// TIA Portal project "FactoryIO_Template_S7-1200_V14" (V14)
// Vorlageprojekt für das Buch mit Zielsystem S7-1200

(* hardware
DEVICE "S7-1200-Station_1"  S7-1200 Station
   slot 0: "Baugruppenträger_0"  Rack  V1.0
   slot 1: "PLC_1"  CPU 1211C DC/DC/DC  6ES7 211-1AE40-0XB0  V4.1
*)

// ===== PLC "PLC_1"  CPU 1211C DC/DC/DC =====

VAR_GLOBAL   // PLC tag table "Standard-Variablentabelle"
   "Clock_Byte" AT %MB85 : Byte;
   "Clock_10Hz" AT %M85.0 : Bool;
   "Clock_5Hz" AT %M85.1 : Bool;
   "Clock_2.5Hz" AT %M85.2 : Bool;
   "Clock_2Hz" AT %M85.3 : Bool;
   "Clock_1.25Hz" AT %M85.4 : Bool;
   "Clock_1Hz" AT %M85.5 : Bool;
   "Clock_0.625Hz" AT %M85.6 : Bool;
   "Clock_0.5Hz" AT %M85.7 : Bool;
   "System_Byte" AT %MB1 : Byte;
   "FirstScan" AT %M1.0 : Bool;
   "DiagStatusUpdate" AT %M1.1 : Bool;
   "AlwaysTRUE" AT %M1.2 : Bool;
   "AlwaysFALSE" AT %M1.3 : Bool;
   "System_Byte(1)" AT %MB1 : Byte;
END_VAR

VAR_GLOBAL   // PLC tag table "Inputs"
   "DI_Item at entry" AT %I0.0 : Bool;
   "DI_Item at exit" AT %I0.1 : Bool;
   "DI_Moving X" AT %I0.2 : Bool;
   "DI_Moving Z" AT %I0.3 : Bool;
   "DI_Item detected" AT %I0.4 : Bool;
   "DI_Start" AT %I0.5 : Bool;
   "DI_Reset" AT %I0.6 : Bool;
   "DI_Stop" AT %I0.7 : Bool;
   "DI_Emergency stop" AT %I1.0 : Bool;
   "DI_Auto" AT %I1.1 : Bool;
   "DI_FACTORY I/O (Running)" AT %I1.2 : Bool;
END_VAR

VAR_GLOBAL   // PLC tag table "Outputs"
   "DO_Entry conveyor" AT %Q0.0 : Bool;
   "DO_Exit conveyor" AT %Q0.1 : Bool;
   "DO_Move X" AT %Q0.2 : Bool;
   "DO_Move Z" AT %Q0.3 : Bool;
   "DO_Grab" AT %Q0.4 : Bool;
   "DO_Start light" AT %Q0.5 : Bool;
   "DO_Reset light" AT %Q0.6 : Bool;
   "DO_Stop light" AT %Q0.7 : Bool;
   "DO_Counter" AT %QD30 : DInt;
END_VAR

// folder: Errors[ER]

DATA_BLOCK "ER_DB_Errors"   // DB8
{ S7_Optimized_Access := 'TRUE' }
VERSION : 0.1
   VAR
      EmergencyButton : Bool;
   END_VAR
BEGIN
END_DATA_BLOCK

// folder: Hardware[HW]

DATA_BLOCK "HW_DB_Signals"   // DB1
{ S7_Optimized_Access := 'TRUE' }
VERSION : 0.1
   VAR
      "Item at entry" : Struct
         Memory : Bool;
         Exact : Bool;
      END_STRUCT;
      "Item at exit" : Struct
         Memory : Bool;
         Exact : Bool;
      END_STRUCT;
      "Item at exit - falling" : Struct
         Memory : Bool;
         Exact : Bool;
      END_STRUCT;
      "Counter" : DInt;
      "Item detected" : Struct
         Memory : Bool;
         Exact : Bool;
      END_STRUCT;
   END_VAR
BEGIN
END_DATA_BLOCK

DATA_BLOCK "HW_DB_DOutputs"   // DB10
{ S7_Optimized_Access := 'TRUE' }
VERSION : 0.1
   VAR
      EntryConveyor : Bool;
      ExitConveyor : Bool;
      MoveX : Bool;
      MoveZ : Bool;
      Grab : Bool;
   END_VAR
BEGIN
END_DATA_BLOCK

// folder: Management[MG]

DATA_BLOCK "MG_DB_ModeSelection"   // DB7
{ S7_Optimized_Access := 'TRUE' }
VERSION : 0.1
   VAR
      Auto : Bool;
      Manual : Bool;
      GlobError : Bool;
   END_VAR
BEGIN
END_DATA_BLOCK

// folder: System blocks/Program resources

DATA_BLOCK "LG_FC_Timer1"   // DB2
{ S7_Optimized_Access := 'TRUE' }
AUTHOR : Simatic
FAMILY : IEC
NAME : IEC_TMR
VERSION : 1.0
// stored: InstanceOfName IEC_TIMER
"IEC_TIMER"
BEGIN
END_DATA_BLOCK

DATA_BLOCK "LG_FC_StartMowivng2"   // DB3
{ S7_Optimized_Access := 'TRUE' }
AUTHOR : Simatic
FAMILY : IEC
NAME : IEC_TMR
VERSION : 1.0
// stored: InstanceOfName IEC_TIMER
"IEC_TIMER"
BEGIN
END_DATA_BLOCK

DATA_BLOCK "LG_FC_MoveEntryConveyor1"   // DB4
{ S7_Optimized_Access := 'TRUE' }
AUTHOR : Simatic
FAMILY : IEC
NAME : IEC_TMR
VERSION : 1.0
// stored: InstanceOfName IEC_TIMER
"IEC_TIMER"
BEGIN
END_DATA_BLOCK

DATA_BLOCK "LG_FC_StartMoving3"   // DB5
{ S7_Optimized_Access := 'TRUE' }
AUTHOR : Simatic
FAMILY : IEC
NAME : IEC_TMR
VERSION : 1.0
// stored: InstanceOfName IEC_TIMER
"IEC_TIMER"
BEGIN
END_DATA_BLOCK

DATA_BLOCK "LG_FC_StartMoving4"   // DB6
{ S7_Optimized_Access := 'TRUE' }
AUTHOR : Simatic
FAMILY : IEC
NAME : IEC_TMR
VERSION : 1.0
// stored: InstanceOfName IEC_TIMER
"IEC_TIMER"
BEGIN
END_DATA_BLOCK

DATA_BLOCK "LG_DB_TimerX"   // DB9
{ S7_Optimized_Access := 'TRUE' }
AUTHOR : Simatic
FAMILY : IEC
NAME : IEC_TMR
VERSION : 1.0
// stored: InstanceOfName IEC_TIMER
"IEC_TIMER"
BEGIN
END_DATA_BLOCK

DATA_BLOCK "LGFC_TimerY"   // DB11
{ S7_Optimized_Access := 'TRUE' }
AUTHOR : Simatic
FAMILY : IEC
NAME : IEC_TMR
VERSION : 1.0
// stored: InstanceOfName IEC_TIMER
"IEC_TIMER"
BEGIN
END_DATA_BLOCK

// folder: (top level)

FUNCTION "MHJ-PLC-Lab-Function-S71200" : Void   // FC9000, SCL
{ S7_Optimized_Access := 'TRUE' }
VERSION : 0.1
   VAR_TEMP
      rdTimeReturn : Int;
      outputTime : DTL;
      SyncVal : Byte;
      forVal : Int;
      forVal_2 : Int;
      Value : Byte;
   END_VAR
   VAR CONSTANT
      CompVal : Byte := 16#34;
      Value_01 : Byte := 16#11;
      Value_01_DW : DWord := 16#A165_D992;
      Value_02_DW : DWord := 16#58BE_4401;
   END_VAR
BEGIN

   #Value:=PEEK(area := 16#82,
        dbNumber := 0,
        byteOffset := 511);
   #Value := #Value + 1;

   POKE(area := 16#82,
        dbNumber := 0,
        byteOffset := 511,
        value := #Value);

   POKE(area:=16#81,
        dbNumber:=0,
        byteOffset:=1016,
        value:=#Value_01_DW);
   POKE(area := 16#81,
        dbNumber := 0,
        byteOffset := 1020,
        value := #Value_02_DW);

   POKE(area := 16#81,
        dbNumber := 0,
        byteOffset := 511,
        value := B#16#00);

   FOR #forVal := 0 TO 120 DO
       FOR #forVal_2:=0 TO 10 DO
           #rdTimeReturn:=RD_SYS_T(#outputTime);
           #rdTimeReturn := WR_SYS_T(#outputTime);
           #rdTimeReturn := RD_SYS_T(#outputTime);
           #rdTimeReturn := WR_SYS_T(#outputTime);
       END_FOR;
       #SyncVal:= PEEK(area := 16#81,
                      dbNumber := 0,
                      byteOffset := 511);
       IF #SyncVal = #CompVal THEN
          GOTO M_1;
       END_IF;
   END_FOR;
   RETURN;

   M_1:
   POKE(area := 16#81,
        dbNumber := 0,
        byteOffset := 511,
        value := B#16#0);
END_FUNCTION

ORGANIZATION_BLOCK "Main"   // OB1, LAD, ProgramCycle
TITLE = "Main Program Sweep (Cycle)"
{ S7_Optimized_Access := 'TRUE' }
VERSION : 0.1
   VAR_INPUT
      Initial_Call : Bool;   // Initial call of this OB
      Remanence : Bool;   // =True, if remanent data are available
   END_VAR
BEGIN

REGION Network 1: Konnektierungsbaustein für PLC-Lab
   // Im Netzwerk 1 wird der Konnektierungsbaustein für PLC-Lab aufgerufen.
   // Dieser Aufruf darf nicht entfernt werden!
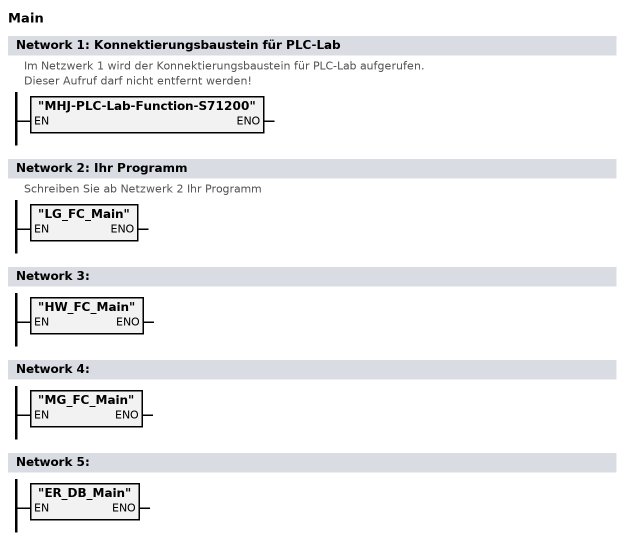
   RUNG wire#powerrail
      "MHJ-PLC-Lab-Function-S71200"()
   END_RUNG
   // the same network as SCL:
   "MHJ-PLC-Lab-Function-S71200"();
END_REGION

REGION Network 2: Ihr Programm
   // Schreiben Sie ab Netzwerk 2 Ihr Programm
   RUNG wire#powerrail
      "LG_FC_Main"()
   END_RUNG
   // the same network as SCL:
   "LG_FC_Main"();
END_REGION

REGION Network 3
   RUNG wire#powerrail
      "HW_FC_Main"()
   END_RUNG
   // the same network as SCL:
   "HW_FC_Main"();
END_REGION

REGION Network 4
   RUNG wire#powerrail
      "MG_FC_Main"()
   END_RUNG
   // the same network as SCL:
   "MG_FC_Main"();
END_REGION

REGION Network 5
   RUNG wire#powerrail
      "ER_DB_Main"()
   END_RUNG
   // the same network as SCL:
   "ER_DB_Main"();
END_REGION
END_ORGANIZATION_BLOCK

// folder: Errors[ER]

FUNCTION "ER_DB_Main" : Void   // FC13, LAD
{ S7_Optimized_Access := 'TRUE' }
VERSION : 0.1
BEGIN

REGION Network 1
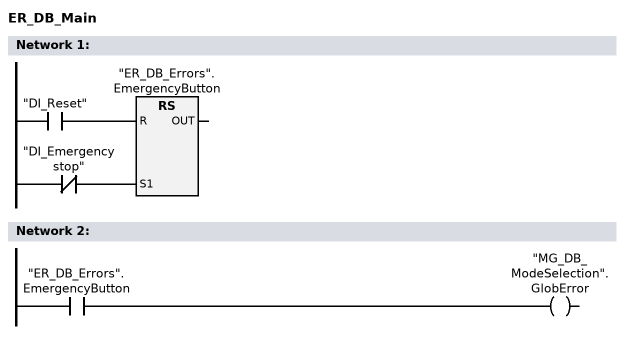
   RUNG wire#powerrail
      Contact( "DI_Reset" )
      S_RS(operand := "ER_DB_Errors".EmergencyButton, s1 := wire#w1)
   END_RUNG
   RUNG wire#powerrail
      I_Contact( "DI_Emergency stop" )
   END_RUNG wire#w1
   // the same network as SCL:
   IF "DI_Reset" THEN
       "ER_DB_Errors".EmergencyButton := FALSE;   // RS flip-flop
   END_IF;
   IF NOT "DI_Emergency stop" THEN "ER_DB_Errors".EmergencyButton := TRUE; END_IF;
END_REGION

REGION Network 2
   RUNG wire#powerrail
      Contact( "ER_DB_Errors".EmergencyButton )
      Coil( "MG_DB_ModeSelection".GlobError )
   END_RUNG
   // the same network as SCL:
   "MG_DB_ModeSelection".GlobError := "ER_DB_Errors".EmergencyButton;
END_REGION
END_FUNCTION

// folder: Hardware[HW]

FUNCTION "HW_FC_RisingSignal" : Void   // FC1, LAD
{ S7_Optimized_Access := 'TRUE' }
VERSION : 0.1
   VAR_INPUT
      I_Signal : Bool;
   END_VAR
   VAR_OUTPUT
      O_Exact : Bool;
   END_VAR
   VAR_IN_OUT
      IO_Memory : Bool;
   END_VAR
   VAR_TEMP   // added for the SCL form of the ladder/FBD networks
      _w1 : Bool;
   END_VAR
BEGIN

REGION Network 1
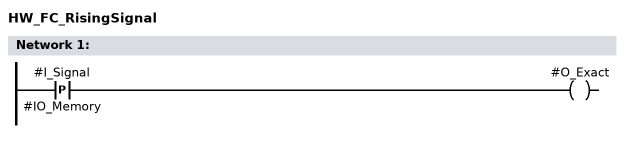
   RUNG wire#powerrail
      P_Contact(operand := #I_Signal, bit := #IO_Memory)
      Coil( #O_Exact )
   END_RUNG
   // the same network as SCL:
   #_w1 := #I_Signal AND NOT #IO_Memory;   // rising edge of #I_Signal
   #IO_Memory := #I_Signal;
   #O_Exact := #_w1;
END_REGION
END_FUNCTION

FUNCTION "HW_FC_FallingSignal" : Void   // FC2, LAD
{ S7_Optimized_Access := 'TRUE' }
VERSION : 0.1
   VAR_INPUT
      I_Signal : Bool;
   END_VAR
   VAR_OUTPUT
      O_Exact : Bool;
   END_VAR
   VAR_IN_OUT
      IO_Memory : Bool;
   END_VAR
   VAR_TEMP   // added for the SCL form of the ladder/FBD networks
      _w1 : Bool;
   END_VAR
BEGIN

REGION Network 1
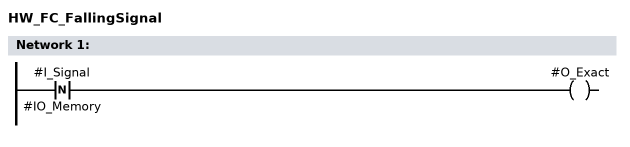
   RUNG wire#powerrail
      N_Contact(operand := #I_Signal, bit := #IO_Memory)
      Coil( #O_Exact )
   END_RUNG
   // the same network as SCL:
   #_w1 := NOT #I_Signal AND #IO_Memory;   // falling edge of #I_Signal
   #IO_Memory := #I_Signal;
   #O_Exact := #_w1;
END_REGION
END_FUNCTION

FUNCTION "HW_FC_Sensors" : Void   // FC3, LAD
{ S7_Optimized_Access := 'TRUE' }
VERSION : 0.1
BEGIN

REGION Network 1
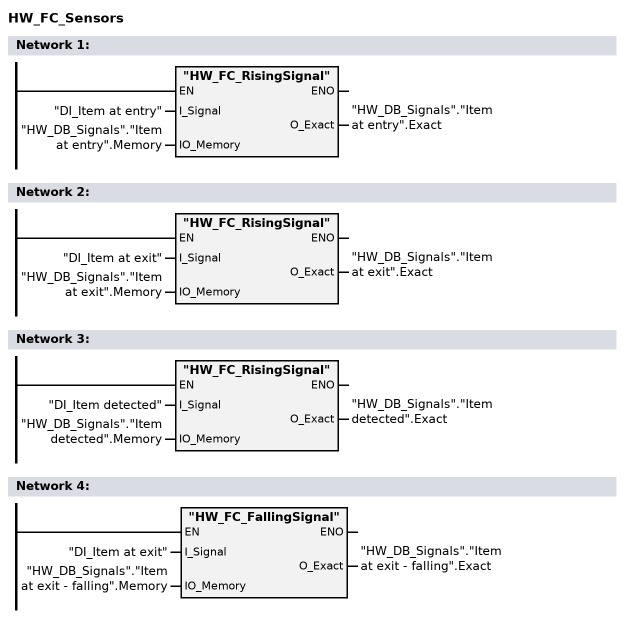
   RUNG wire#powerrail
      "HW_FC_RisingSignal"(I_Signal := "DI_Item at entry", IO_Memory := "HW_DB_Signals"."Item at entry".Memory, O_Exact => "HW_DB_Signals"."Item at entry".Exact)
   END_RUNG
   // the same network as SCL:
   "HW_FC_RisingSignal"(I_Signal := "DI_Item at entry",
                        IO_Memory := "HW_DB_Signals"."Item at entry".Memory,
                        O_Exact => "HW_DB_Signals"."Item at entry".Exact);
END_REGION

REGION Network 2
   RUNG wire#powerrail
      "HW_FC_RisingSignal"(I_Signal := "DI_Item at exit", IO_Memory := "HW_DB_Signals"."Item at exit".Memory, O_Exact => "HW_DB_Signals"."Item at exit".Exact)
   END_RUNG
   // the same network as SCL:
   "HW_FC_RisingSignal"(I_Signal := "DI_Item at exit",
                        IO_Memory := "HW_DB_Signals"."Item at exit".Memory,
                        O_Exact => "HW_DB_Signals"."Item at exit".Exact);
END_REGION

REGION Network 3
   RUNG wire#powerrail
      "HW_FC_RisingSignal"(I_Signal := "DI_Item detected", IO_Memory := "HW_DB_Signals"."Item detected".Memory, O_Exact => "HW_DB_Signals"."Item detected".Exact)
   END_RUNG
   // the same network as SCL:
   "HW_FC_RisingSignal"(I_Signal := "DI_Item detected",
                        IO_Memory := "HW_DB_Signals"."Item detected".Memory,
                        O_Exact => "HW_DB_Signals"."Item detected".Exact);
END_REGION

REGION Network 4
   RUNG wire#powerrail
      "HW_FC_FallingSignal"(I_Signal := "DI_Item at exit", IO_Memory := "HW_DB_Signals"."Item at exit - falling".Memory, O_Exact => "HW_DB_Signals"."Item at exit - falling".Exact)
   END_RUNG
   // the same network as SCL:
   "HW_FC_FallingSignal"(I_Signal := "DI_Item at exit",
                         IO_Memory := "HW_DB_Signals"."Item at exit - falling".Memory,
                         O_Exact => "HW_DB_Signals"."Item at exit - falling".Exact);
END_REGION
END_FUNCTION

FUNCTION "HW_FC_Counting" : Void   // FC5, LAD
{ S7_Optimized_Access := 'TRUE' }
VERSION : 0.1
BEGIN

REGION Network 1
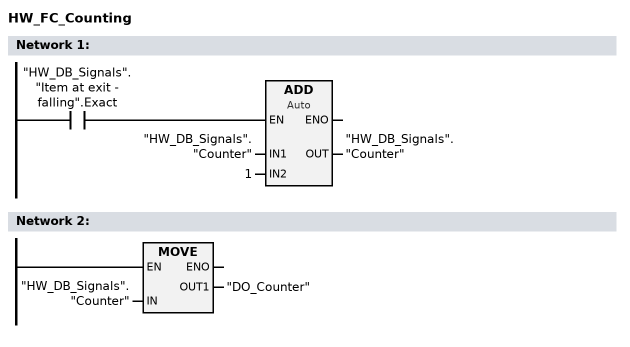
   RUNG wire#powerrail
      Contact( "HW_DB_Signals"."Item at exit - falling".Exact )
      Add(in1 := "HW_DB_Signals"."Counter", in2 := 1, out => "HW_DB_Signals"."Counter")
   END_RUNG
   // the same network as SCL:
   IF "HW_DB_Signals"."Item at exit - falling".Exact THEN
       "HW_DB_Signals"."Counter" := "HW_DB_Signals"."Counter" + 1;
   END_IF;
END_REGION

REGION Network 2
   RUNG wire#powerrail
      Move(in := "HW_DB_Signals"."Counter", out1 => "DO_Counter")
   END_RUNG
   // the same network as SCL:
   "DO_Counter" := "HW_DB_Signals"."Counter";
END_REGION
END_FUNCTION

FUNCTION "HW_FC_Main" : Void   // FC7, LAD
{ S7_Optimized_Access := 'TRUE' }
VERSION : 0.1
BEGIN

REGION Network 1
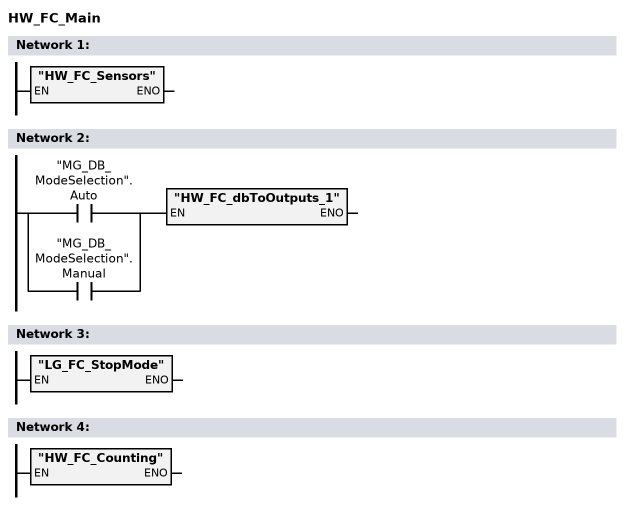
   RUNG wire#powerrail
      "HW_FC_Sensors"()
   END_RUNG
   // the same network as SCL:
   "HW_FC_Sensors"();
END_REGION

REGION Network 2
   RUNG wire#powerrail
      Contact( "MG_DB_ModeSelection".Auto )
      wire#w1
      "HW_FC_dbToOutputs_1"()
   END_RUNG
   RUNG wire#powerrail
      Contact( "MG_DB_ModeSelection".Manual )
   END_RUNG wire#w1
   // the same network as SCL:
   IF "MG_DB_ModeSelection".Auto OR "MG_DB_ModeSelection".Manual THEN "HW_FC_dbToOutputs_1"(); END_IF;
END_REGION

REGION Network 3
   RUNG wire#powerrail
      "LG_FC_StopMode"()
   END_RUNG
   // the same network as SCL:
   "LG_FC_StopMode"();
END_REGION

REGION Network 4
   RUNG wire#powerrail
      "HW_FC_Counting"()
   END_RUNG
   // the same network as SCL:
   "HW_FC_Counting"();
END_REGION
END_FUNCTION

FUNCTION "HW_FC_dbToOutputs_1" : Void   // FC14, LAD
{ S7_Optimized_Access := 'TRUE' }
VERSION : 0.1
BEGIN

REGION Network 1
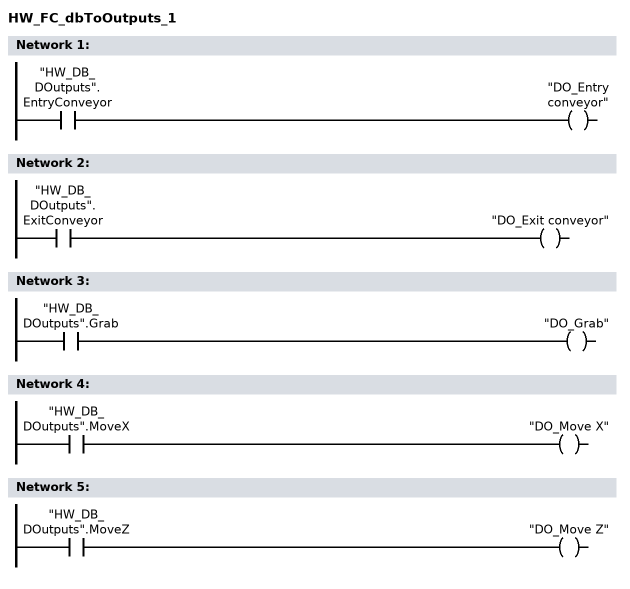
   RUNG wire#powerrail
      Contact( "HW_DB_DOutputs".EntryConveyor )
      Coil( "DO_Entry conveyor" )
   END_RUNG
   // the same network as SCL:
   "DO_Entry conveyor" := "HW_DB_DOutputs".EntryConveyor;
END_REGION

REGION Network 2
   RUNG wire#powerrail
      Contact( "HW_DB_DOutputs".ExitConveyor )
      Coil( "DO_Exit conveyor" )
   END_RUNG
   // the same network as SCL:
   "DO_Exit conveyor" := "HW_DB_DOutputs".ExitConveyor;
END_REGION

REGION Network 3
   RUNG wire#powerrail
      Contact( "HW_DB_DOutputs".Grab )
      Coil( "DO_Grab" )
   END_RUNG
   // the same network as SCL:
   "DO_Grab" := "HW_DB_DOutputs".Grab;
END_REGION

REGION Network 4
   RUNG wire#powerrail
      Contact( "HW_DB_DOutputs".MoveX )
      Coil( "DO_Move X" )
   END_RUNG
   // the same network as SCL:
   "DO_Move X" := "HW_DB_DOutputs".MoveX;
END_REGION

REGION Network 5
   RUNG wire#powerrail
      Contact( "HW_DB_DOutputs".MoveZ )
      Coil( "DO_Move Z" )
   END_RUNG
   // the same network as SCL:
   "DO_Move Z" := "HW_DB_DOutputs".MoveZ;
END_REGION
END_FUNCTION

// folder: Logical[LG]

FUNCTION "LG_FC_Main" : Void   // FC4, LAD
{ S7_Optimized_Access := 'TRUE' }
VERSION : 0.1
BEGIN

REGION Network 1
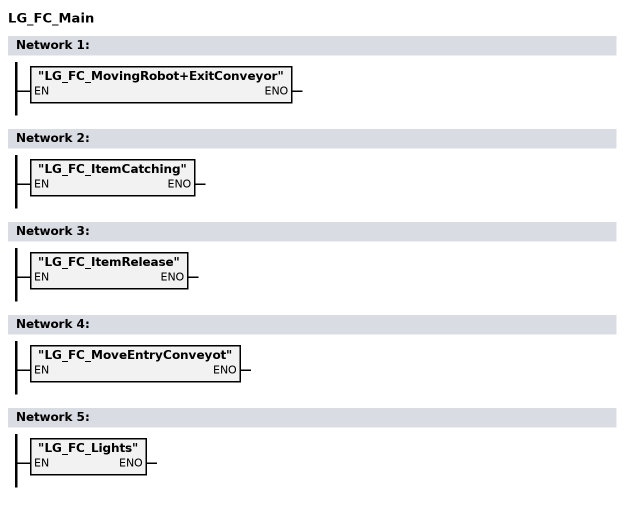
   RUNG wire#powerrail
      "LG_FC_MovingRobot+ExitConveyor"()
   END_RUNG
   // the same network as SCL:
   "LG_FC_MovingRobot+ExitConveyor"();
END_REGION

REGION Network 2
   RUNG wire#powerrail
      "LG_FC_ItemCatching"()
   END_RUNG
   // the same network as SCL:
   "LG_FC_ItemCatching"();
END_REGION

REGION Network 3
   RUNG wire#powerrail
      "LG_FC_ItemRelease"()
   END_RUNG
   // the same network as SCL:
   "LG_FC_ItemRelease"();
END_REGION

REGION Network 4
   RUNG wire#powerrail
      "LG_FC_MoveEntryConveyot"()
   END_RUNG
   // the same network as SCL:
   "LG_FC_MoveEntryConveyot"();
END_REGION

REGION Network 5
   RUNG wire#powerrail
      "LG_FC_Lights"()
   END_RUNG
   // the same network as SCL:
   "LG_FC_Lights"();
END_REGION
END_FUNCTION

FUNCTION "LG_FC_ItemCatching" : Void   // FC6, LAD
{ S7_Optimized_Access := 'TRUE' }
VERSION : 0.1
BEGIN

REGION Network 1
   // Łapanie przedmiotu
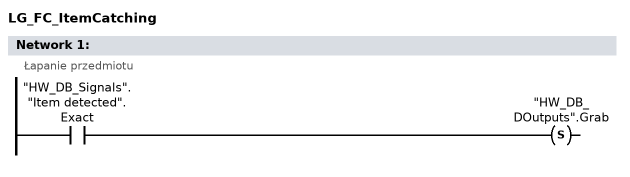
   RUNG wire#powerrail
      Contact( "HW_DB_Signals"."Item detected".Exact )
      S_Coil( "HW_DB_DOutputs".Grab )
   END_RUNG
   // the same network as SCL:
   IF "HW_DB_Signals"."Item detected".Exact THEN "HW_DB_DOutputs".Grab := TRUE; END_IF;
END_REGION
END_FUNCTION

FUNCTION "LG_FC_ItemRelease" : Void   // FC8, LAD
{ S7_Optimized_Access := 'TRUE' }
VERSION : 0.1
BEGIN

REGION Network 1
   // Puszczanie przedmiotu
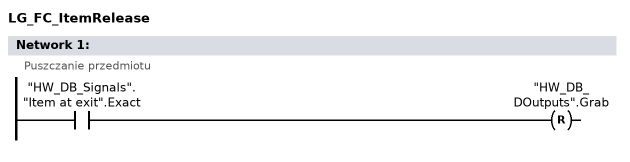
   RUNG wire#powerrail
      Contact( "HW_DB_Signals"."Item at exit".Exact )
      R_Coil( "HW_DB_DOutputs".Grab )
   END_RUNG
   // the same network as SCL:
   IF "HW_DB_Signals"."Item at exit".Exact THEN "HW_DB_DOutputs".Grab := FALSE; END_IF;
END_REGION
END_FUNCTION

FUNCTION "LG_FC_MovingRobot+ExitConveyor" : Void   // FC9, LAD
{ S7_Optimized_Access := 'TRUE' }
VERSION : 0.1
BEGIN

REGION Network 1
   // Przenoszenie cz. 1/4 - Ruszenie "Z" w dół
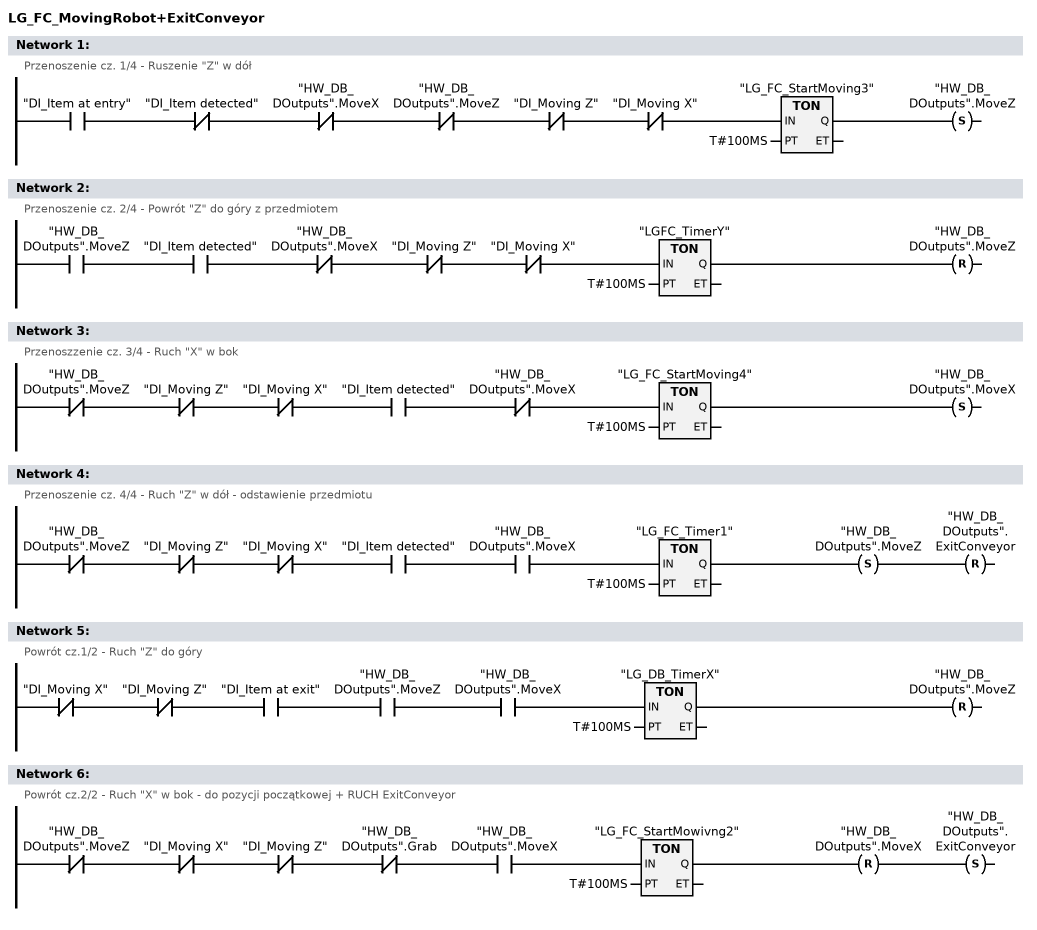
   "LG_FC_StartMoving3".TON(IN := "DI_Item at entry" AND NOT "DI_Item detected" AND NOT "HW_DB_DOutputs".MoveX AND NOT "HW_DB_DOutputs".MoveZ AND NOT "DI_Moving Z" AND NOT "DI_Moving X",
                           PT := T#100MS);
   IF "LG_FC_StartMoving3".Q THEN "HW_DB_DOutputs".MoveZ := TRUE; END_IF;
END_REGION

REGION Network 2
   // Przenoszenie cz. 2/4 - Powrót "Z" do góry z przedmiotem
   "LGFC_TimerY".TON(IN := "HW_DB_DOutputs".MoveZ AND "DI_Item detected" AND NOT "HW_DB_DOutputs".MoveX AND NOT "DI_Moving Z" AND NOT "DI_Moving X",
                     PT := T#100MS);
   IF "LGFC_TimerY".Q THEN "HW_DB_DOutputs".MoveZ := FALSE; END_IF;
END_REGION

REGION Network 3
   // Przenoszzenie cz. 3/4 - Ruch "X" w bok
   "LG_FC_StartMoving4".TON(IN := NOT "HW_DB_DOutputs".MoveZ AND NOT "DI_Moving Z" AND NOT "DI_Moving X" AND "DI_Item detected" AND NOT "HW_DB_DOutputs".MoveX,
                           PT := T#100MS);
   IF "LG_FC_StartMoving4".Q THEN "HW_DB_DOutputs".MoveX := TRUE; END_IF;
END_REGION

REGION Network 4
   // Przenoszenie cz. 4/4 - Ruch "Z" w dół - odstawienie przedmiotu
   "LG_FC_Timer1".TON(IN := NOT "HW_DB_DOutputs".MoveZ AND NOT "DI_Moving Z" AND NOT "DI_Moving X" AND "DI_Item detected" AND "HW_DB_DOutputs".MoveX,
                      PT := T#100MS);
   IF "LG_FC_Timer1".Q THEN
       "HW_DB_DOutputs".MoveZ := TRUE;
       "HW_DB_DOutputs".ExitConveyor := FALSE;
   END_IF;
END_REGION

REGION Network 5
   // Powrót cz.1/2 - Ruch "Z" do góry
   "LG_DB_TimerX".TON(IN := NOT "DI_Moving X" AND NOT "DI_Moving Z" AND "DI_Item at exit" AND "HW_DB_DOutputs".MoveZ AND "HW_DB_DOutputs".MoveX,
                      PT := T#100MS);
   IF "LG_DB_TimerX".Q THEN "HW_DB_DOutputs".MoveZ := FALSE; END_IF;
END_REGION

REGION Network 6
   // Powrót cz.2/2 - Ruch "X" w bok - do pozycji początkowej + RUCH ExitConveyor
   "LG_FC_StartMowivng2".TON(IN := NOT "HW_DB_DOutputs".MoveZ AND NOT "DI_Moving X" AND NOT "DI_Moving Z" AND NOT "HW_DB_DOutputs".Grab AND "HW_DB_DOutputs".MoveX,
                           PT := T#100MS);
   IF "LG_FC_StartMowivng2".Q THEN
       "HW_DB_DOutputs".MoveX := FALSE;
       "HW_DB_DOutputs".ExitConveyor := TRUE;
   END_IF;
END_REGION
END_FUNCTION

FUNCTION "LG_FC_MoveEntryConveyot" : Void   // FC10, LAD
{ S7_Optimized_Access := 'TRUE' }
VERSION : 0.1
BEGIN

REGION Network 1
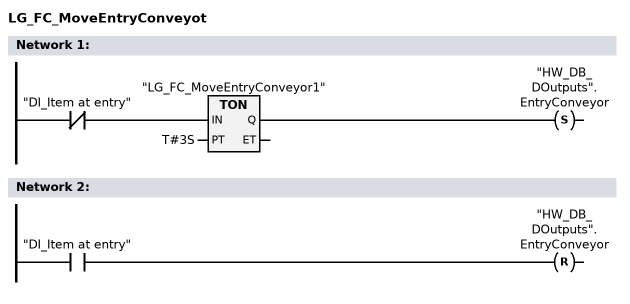
   "LG_FC_MoveEntryConveyor1".TON(IN := NOT "DI_Item at entry", PT := T#3S);
   IF "LG_FC_MoveEntryConveyor1".Q THEN "HW_DB_DOutputs".EntryConveyor := TRUE; END_IF;
END_REGION

REGION Network 2
   RUNG wire#powerrail
      Contact( "DI_Item at entry" )
      R_Coil( "HW_DB_DOutputs".EntryConveyor )
   END_RUNG
   // the same network as SCL:
   IF "DI_Item at entry" THEN "HW_DB_DOutputs".EntryConveyor := FALSE; END_IF;
END_REGION
END_FUNCTION

FUNCTION "LG_FC_Lights" : Void   // FC12, LAD
{ S7_Optimized_Access := 'TRUE' }
VERSION : 0.1
BEGIN

REGION Network 1
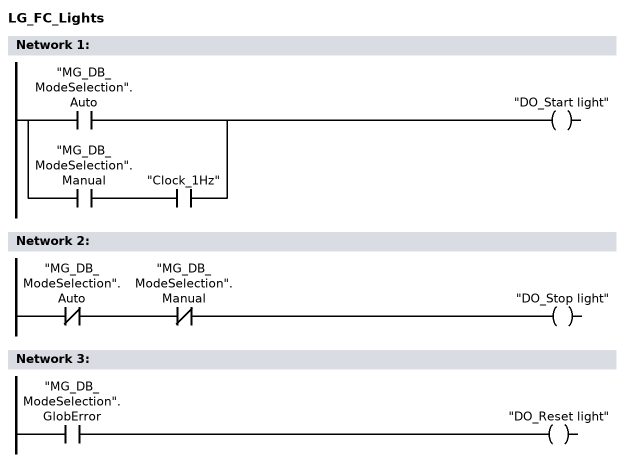
   RUNG wire#powerrail
      Contact( "MG_DB_ModeSelection".Auto )
      wire#w1
      Coil( "DO_Start light" )
   END_RUNG
   RUNG wire#powerrail
      Contact( "MG_DB_ModeSelection".Manual )
      Contact( "Clock_1Hz" )
   END_RUNG wire#w1
   // the same network as SCL:
   "DO_Start light" := "MG_DB_ModeSelection".Auto OR ("MG_DB_ModeSelection".Manual AND "Clock_1Hz");
END_REGION

REGION Network 2
   RUNG wire#powerrail
      I_Contact( "MG_DB_ModeSelection".Auto )
      I_Contact( "MG_DB_ModeSelection".Manual )
      Coil( "DO_Stop light" )
   END_RUNG
   // the same network as SCL:
   "DO_Stop light" := NOT "MG_DB_ModeSelection".Auto AND NOT "MG_DB_ModeSelection".Manual;
END_REGION

REGION Network 3
   RUNG wire#powerrail
      Contact( "MG_DB_ModeSelection".GlobError )
      Coil( "DO_Reset light" )
   END_RUNG
   // the same network as SCL:
   "DO_Reset light" := "MG_DB_ModeSelection".GlobError;
END_REGION
END_FUNCTION

FUNCTION "LG_FC_StopMode" : Void   // FC15, LAD
{ S7_Optimized_Access := 'TRUE' }
VERSION : 0.1
BEGIN

REGION Network 1
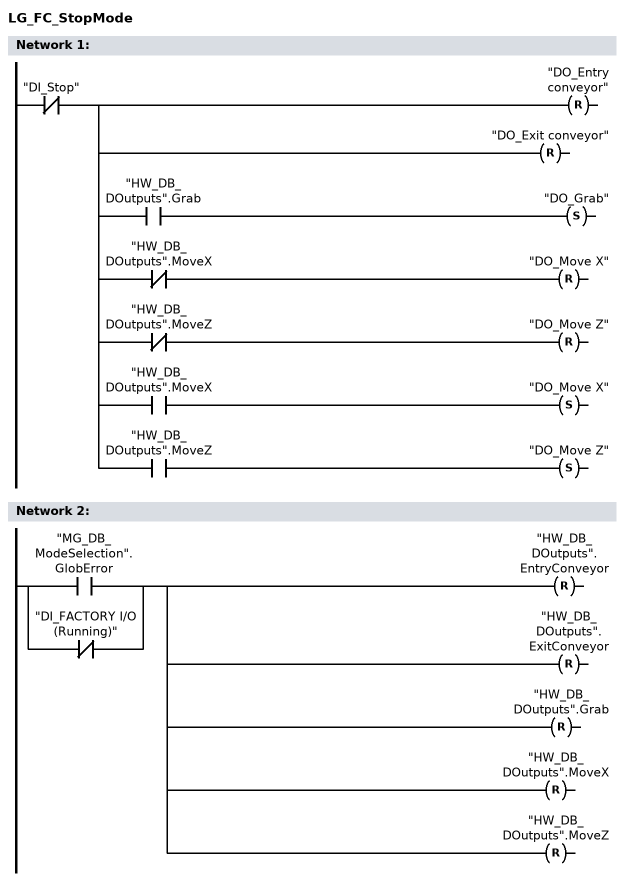
   RUNG wire#powerrail
      I_Contact( "DI_Stop" )
      wire#w1
      R_Coil( "DO_Entry conveyor" )
   END_RUNG
   RUNG wire#w1
      R_Coil( "DO_Exit conveyor" )
   END_RUNG
   RUNG wire#w1
      Contact( "HW_DB_DOutputs".Grab )
      S_Coil( "DO_Grab" )
   END_RUNG
   RUNG wire#w1
      I_Contact( "HW_DB_DOutputs".MoveX )
      R_Coil( "DO_Move X" )
   END_RUNG
   RUNG wire#w1
      I_Contact( "HW_DB_DOutputs".MoveZ )
      R_Coil( "DO_Move Z" )
   END_RUNG
   RUNG wire#w1
      Contact( "HW_DB_DOutputs".MoveX )
      S_Coil( "DO_Move X" )
   END_RUNG
   RUNG wire#w1
      Contact( "HW_DB_DOutputs".MoveZ )
      S_Coil( "DO_Move Z" )
   END_RUNG
   // the same network as SCL:
   IF NOT "DI_Stop" THEN
       "DO_Entry conveyor" := FALSE;
       "DO_Exit conveyor" := FALSE;
   END_IF;
   IF NOT "DI_Stop" AND "HW_DB_DOutputs".Grab THEN "DO_Grab" := TRUE; END_IF;
   IF NOT "DI_Stop" AND NOT "HW_DB_DOutputs".MoveX THEN "DO_Move X" := FALSE; END_IF;
   IF NOT "DI_Stop" AND NOT "HW_DB_DOutputs".MoveZ THEN "DO_Move Z" := FALSE; END_IF;
   IF NOT "DI_Stop" AND "HW_DB_DOutputs".MoveX THEN "DO_Move X" := TRUE; END_IF;
   IF NOT "DI_Stop" AND "HW_DB_DOutputs".MoveZ THEN "DO_Move Z" := TRUE; END_IF;
END_REGION

REGION Network 2
   RUNG wire#powerrail
      Contact( "MG_DB_ModeSelection".GlobError )
      wire#w1
      R_Coil( "HW_DB_DOutputs".EntryConveyor )
   END_RUNG
   RUNG wire#powerrail
      I_Contact( "DI_FACTORY I/O (Running)" )
   END_RUNG wire#w1
   RUNG wire#w1
      R_Coil( "HW_DB_DOutputs".ExitConveyor )
   END_RUNG
   RUNG wire#w1
      R_Coil( "HW_DB_DOutputs".Grab )
   END_RUNG
   RUNG wire#w1
      R_Coil( "HW_DB_DOutputs".MoveX )
   END_RUNG
   RUNG wire#w1
      R_Coil( "HW_DB_DOutputs".MoveZ )
   END_RUNG
   // the same network as SCL:
   IF "MG_DB_ModeSelection".GlobError OR NOT "DI_FACTORY I/O (Running)" THEN
       "HW_DB_DOutputs".EntryConveyor := FALSE;
       "HW_DB_DOutputs".ExitConveyor := FALSE;
       "HW_DB_DOutputs".Grab := FALSE;
       "HW_DB_DOutputs".MoveX := FALSE;
       "HW_DB_DOutputs".MoveZ := FALSE;
   END_IF;
END_REGION
END_FUNCTION

// folder: Management[MG]

FUNCTION "MG_FC_Main" : Void   // FC11, LAD
{ S7_Optimized_Access := 'TRUE' }
VERSION : 0.1
BEGIN

REGION Network 1
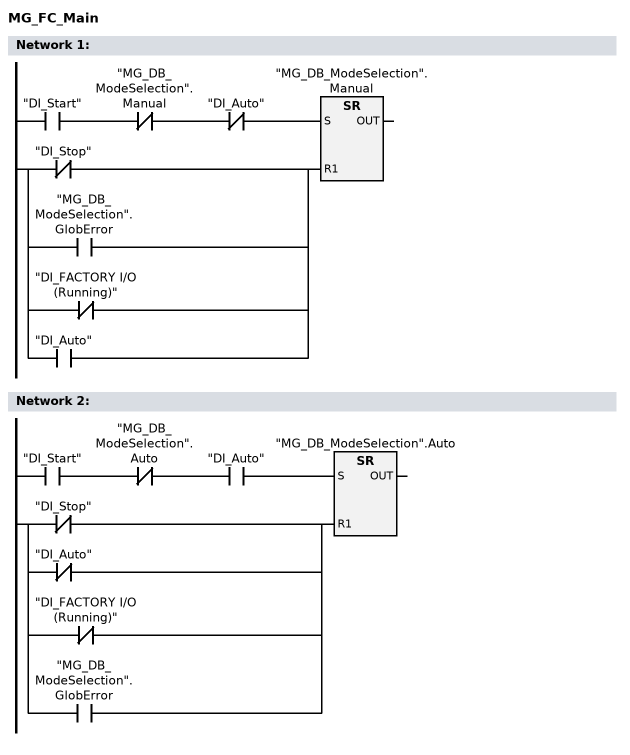
   RUNG wire#powerrail
      Contact( "DI_Start" )
      I_Contact( "MG_DB_ModeSelection".Manual )
      I_Contact( "DI_Auto" )
      S_SR(operand := "MG_DB_ModeSelection".Manual, r1 := wire#w1)
   END_RUNG
   RUNG wire#powerrail
      I_Contact( "DI_Stop" )
   END_RUNG wire#w1
   RUNG wire#powerrail
      Contact( "MG_DB_ModeSelection".GlobError )
   END_RUNG wire#w1
   RUNG wire#powerrail
      I_Contact( "DI_FACTORY I/O (Running)" )
   END_RUNG wire#w1
   RUNG wire#powerrail
      Contact( "DI_Auto" )
   END_RUNG wire#w1
   // the same network as SCL:
   IF "DI_Start" AND NOT "MG_DB_ModeSelection".Manual AND NOT "DI_Auto" THEN
       "MG_DB_ModeSelection".Manual := TRUE;   // SR flip-flop
   END_IF;
   IF NOT "DI_Stop" OR "MG_DB_ModeSelection".GlobError OR NOT "DI_FACTORY I/O (Running)" OR "DI_Auto" THEN
       "MG_DB_ModeSelection".Manual := FALSE;
   END_IF;
END_REGION

REGION Network 2
   RUNG wire#powerrail
      Contact( "DI_Start" )
      I_Contact( "MG_DB_ModeSelection".Auto )
      Contact( "DI_Auto" )
      S_SR(operand := "MG_DB_ModeSelection".Auto, r1 := wire#w1)
   END_RUNG
   RUNG wire#powerrail
      I_Contact( "DI_Stop" )
   END_RUNG wire#w1
   RUNG wire#powerrail
      I_Contact( "DI_Auto" )
   END_RUNG wire#w1
   RUNG wire#powerrail
      I_Contact( "DI_FACTORY I/O (Running)" )
   END_RUNG wire#w1
   RUNG wire#powerrail
      Contact( "MG_DB_ModeSelection".GlobError )
   END_RUNG wire#w1
   // the same network as SCL:
   IF "DI_Start" AND NOT "MG_DB_ModeSelection".Auto AND "DI_Auto" THEN
       "MG_DB_ModeSelection".Auto := TRUE;   // SR flip-flop
   END_IF;
   IF NOT "DI_Stop" OR NOT "DI_Auto" OR NOT "DI_FACTORY I/O (Running)" OR "MG_DB_ModeSelection".GlobError THEN
       "MG_DB_ModeSelection".Auto := FALSE;
   END_IF;
END_REGION
END_FUNCTION